TYPE ST_DCR_Parameters :
STRUCT
	sampleParameters	: ST_SampleParameters;
	programOptions		: ST_DCR_ProgramOptions;
END_STRUCT
END_TYPE

(* stored: Version 1.1.0.1, ProductVersion 3.1.4024.2
   DUT ST_DCR_Parameters: Id {562880da-b371-4644-98bc-fb98c2f3cbb2} *)
